                                                                                              MoveJ speed 60 deg/s, acceleration 80 deg/s^2 (useActiveTCP=true) feature=Base
                                                                                                Waypoint Waypoint_58: TCP in base x=365.318 y=-268.384 z=96.47 mm, rx=-1.8274 ry=-0.0328 rz=-0.0063 rad; joints [-29.465, -175.579, 2.323, 201.363, 146.436, -157.102] deg
                                                                                                URCap Gripper (Robotiq_Grippers, Robotiq Inc.) dataModel(position=0.0, force=0.0, speed=0.0, positionInDouble=0.0, forceInDouble=0.0, speedInDouble=0.0, slaveIds=[2], blocking=true)
                                                                                                MoveJ speed 60 deg/s, acceleration 80 deg/s^2 (useActiveTCP=true) feature=Base
                                                                                                  Waypoint Waypoint_2: motionParameters(jointSpeed=1.047198 jointAcceleration=1.396263 cartesianSpeed=0.25 cartesianAcceleration=1.2); TCP in base x=280.608 y=-116.08 z=398.046 mm, rx=-2.2371 ry=2.1464 rz=-0.0359 rad; joints [2.971, -88.172, -66.4, 247.256, 90.066, 0.681] deg
                                                                                                  MoveJ speed 60 deg/s, acceleration 80 deg/s^2 (useActiveTCP=true) feature=Base
                                                                                                    Waypoint Waypoint_56: TCP in base x=364.265 y=-116.054 z=192.334 mm, rx=-3.095 ry=0.0588 rz=0.0169 rad; joints [1.825, -110.55, -95.649, 295.749, 92.143, -86.362] deg
                                                                                                    URCap Gripper (Robotiq_Grippers, Robotiq Inc.) dataModel(position=100.0, force=0.0, speed=0.0, positionInDouble=100.0, forceInDouble=0.0, speedInDouble=0.0, slaveIds=[2], blocking=true)
                                                                                                    MoveJ speed 60 deg/s, acceleration 80 deg/s^2 (useActiveTCP=true) feature=Base
                                                                                                      Waypoint Waypoint_57: TCP in base x=364.254 y=-116.07 z=333.901 mm, rx=-3.0957 ry=-0.0405 rz=0.0191 rad; joints [1.801, -106.047, -62.68, 258.123, 92.053, -89.758] deg
                                                                                                      MoveJ speed 60 deg/s, acceleration 80 deg/s^2 (useActiveTCP=true) feature=Base
                                                                                                        Waypoint Waypoint_58: TCP in base x=365.318 y=-268.384 z=96.47 mm, rx=-1.8274 ry=-0.0328 rz=-0.0063 rad; joints [-29.465, -175.579, 2.323, 201.363, 146.436, -157.102] deg
                                                                                                        URCap Gripper (Robotiq_Grippers, Robotiq Inc.) dataModel(position=0.0, force=0.0, speed=0.0, positionInDouble=0.0, forceInDouble=0.0, speedInDouble=0.0, slaveIds=[2], blocking=true)
                                                                                                        MoveJ speed 60 deg/s, acceleration 80 deg/s^2 (useActiveTCP=true) feature=Base
                                                                                                          Waypoint Waypoint_2: motionParameters(jointSpeed=1.047198 jointAcceleration=1.396263 cartesianSpeed=0.25 cartesianAcceleration=1.2); TCP in base x=280.608 y=-116.08 z=398.046 mm, rx=-2.2371 ry=2.1464 rz=-0.0359 rad; joints [2.971, -88.172, -66.4, 247.256, 90.066, 0.681] deg
                                                                                                          Folder Mouvement D2
                                                                                                            MoveJ speed 60 deg/s, acceleration 80 deg/s^2 (useActiveTCP=true) feature=Base
                                                                                                              Waypoint Waypoint_2: motionParameters(jointSpeed=1.047198 jointAcceleration=1.396263 cartesianSpeed=0.25 cartesianAcceleration=1.2); TCP in base x=280.608 y=-116.08 z=398.046 mm, rx=-2.2371 ry=2.1464 rz=-0.0359 rad; joints [2.971, -88.172, -66.4, 247.256, 90.066, 0.681] deg
                                                                                                              MoveJ speed 60 deg/s, acceleration 80 deg/s^2 (useActiveTCP=true) feature=Base
                                                                                                                Waypoint Waypoint_56: TCP in base x=364.265 y=-116.054 z=192.334 mm, rx=-3.095 ry=0.0588 rz=0.0169 rad; joints [1.825, -110.55, -95.649, 295.749, 92.143, -86.362] deg
                                                                                                                URCap Gripper (Robotiq_Grippers, Robotiq Inc.) dataModel(position=100.0, force=0.0, speed=0.0, positionInDouble=100.0, forceInDouble=0.0, speedInDouble=0.0, slaveIds=[2], blocking=true)
                                                                                                                MoveJ speed 60 deg/s, acceleration 80 deg/s^2 (useActiveTCP=true) feature=Base
                                                                                                                  Waypoint Waypoint_57: TCP in base x=364.254 y=-116.07 z=333.901 mm, rx=-3.0957 ry=-0.0405 rz=0.0191 rad; joints [1.801, -106.047, -62.68, 258.123, 92.053, -89.758] deg
                                                                                                                  MoveJ speed 60 deg/s, acceleration 80 deg/s^2 (useActiveTCP=true) feature=Base
                                                                                                                    Waypoint Waypoint_58: TCP in base x=365.318 y=-268.384 z=96.47 mm, rx=-1.8274 ry=-0.0328 rz=-0.0063 rad; joints [-29.465, -175.579, 2.323, 201.363, 146.436, -157.102] deg
                                                                                                                    URCap Gripper (Robotiq_Grippers, Robotiq Inc.) dataModel(position=0.0, force=0.0, speed=0.0, positionInDouble=0.0, forceInDouble=0.0, speedInDouble=0.0, slaveIds=[2], blocking=true)
                                                                                                                    MoveJ speed 60 deg/s, acceleration 80 deg/s^2 (useActiveTCP=true) feature=Base
                                                                                                                      Waypoint Waypoint_2: motionParameters(jointSpeed=1.047198 jointAcceleration=1.396263 cartesianSpeed=0.25 cartesianAcceleration=1.2); TCP in base x=280.608 y=-116.08 z=398.046 mm, rx=-2.2371 ry=2.1464 rz=-0.0359 rad; joints [2.971, -88.172, -66.4, 247.256, 90.066, 0.681] deg
                                                                                                                      MoveJ speed 60 deg/s, acceleration 80 deg/s^2 (useActiveTCP=true) feature=Base
                                                                                                                        Waypoint Waypoint_56: TCP in base x=364.265 y=-116.054 z=192.334 mm, rx=-3.095 ry=0.0588 rz=0.0169 rad; joints [1.825, -110.55, -95.649, 295.749, 92.143, -86.362] deg
                                                                                                                        URCap Gripper (Robotiq_Grippers, Robotiq Inc.) dataModel(position=100.0, force=0.0, speed=0.0, positionInDouble=100.0, forceInDouble=0.0, speedInDouble=0.0, slaveIds=[2], blocking=true)
                                                                                                                        MoveJ speed 60 deg/s, acceleration 80 deg/s^2 (useActiveTCP=true) feature=Base
                                                                                                                          Waypoint Waypoint_57: TCP in base x=364.254 y=-116.07 z=333.901 mm, rx=-3.0957 ry=-0.0405 rz=0.0191 rad; joints [1.801, -106.047, -62.68, 258.123, 92.053, -89.758] deg
                                                                                                                          MoveJ speed 60 deg/s, acceleration 80 deg/s^2 (useActiveTCP=true) feature=Base
                                                                                                                            Waypoint Waypoint_58: TCP in base x=365.318 y=-268.384 z=96.47 mm, rx=-1.8274 ry=-0.0328 rz=-0.0063 rad; joints [-29.465, -175.579, 2.323, 201.363, 146.436, -157.102] deg
                                                                                                                            URCap Gripper (Robotiq_Grippers, Robotiq Inc.) dataModel(position=0.0, force=0.0, speed=0.0, positionInDouble=0.0, forceInDouble=0.0, speedInDouble=0.0, slaveIds=[2], blocking=true)
                                                                                                                            MoveJ speed 60 deg/s, acceleration 80 deg/s^2 (useActiveTCP=true) feature=Base
                                                                                                                              Waypoint Waypoint_2: motionParameters(jointSpeed=1.047198 jointAcceleration=1.396263 cartesianSpeed=0.25 cartesianAcceleration=1.2); TCP in base x=280.608 y=-116.08 z=398.046 mm, rx=-2.2371 ry=2.1464 rz=-0.0359 rad; joints [2.971, -88.172, -66.4, 247.256, 90.066, 0.681] deg
                                                                                                                              MoveJ speed 60 deg/s, acceleration 80 deg/s^2 (useActiveTCP=true) feature=Base
                                                                                                                                Waypoint Waypoint_59: TCP in base x=361.348 y=-116.091 z=193.172 mm, rx=-2.2553 ry=2.1644 rz=0.0052 rad; joints [2.324, -109.416, -97.451, 297.435, 90.248, -0.396] deg
                                                                                                                                URCap Gripper (Robotiq_Grippers, Robotiq Inc.) dataModel(position=100.0, force=0.0, speed=0.0, positionInDouble=100.0, forceInDouble=0.0, speedInDouble=0.0, slaveIds=[2], blocking=true)
                                                                                                                                MoveJ speed 60 deg/s, acceleration 80 deg/s^2 (useActiveTCP=true) feature=Base
                                                                                                                                  Waypoint Waypoint_63: TCP in base x=361.345 y=-116.096 z=193.168 mm, rx=2.0818 ry=2.2845 rz=0.0599 rad; joints [2.646, -108.789, -99.797, 302.251, 89.051, 176.908] deg
                                                                                                                                  URCap Gripper (Robotiq_Grippers, Robotiq Inc.) dataModel(position=0.0, force=0.0, speed=0.0, positionInDouble=0.0, forceInDouble=0.0, speedInDouble=0.0, slaveIds=[2], blocking=true)
                                                                                                                                  MoveJ speed 60 deg/s, acceleration 80 deg/s^2 (useActiveTCP=true) feature=Base
                                                                                                                                    Waypoint Waypoint_2: motionParameters(jointSpeed=1.047198 jointAcceleration=1.396263 cartesianSpeed=0.25 cartesianAcceleration=1.2); TCP in base x=280.608 y=-116.08 z=398.046 mm, rx=-2.2371 ry=2.1464 rz=-0.0359 rad; joints [2.971, -88.172, -66.4, 247.256, 90.066, 0.681] deg
                                                                                                                                    MoveJ speed 60 deg/s, acceleration 80 deg/s^2 (useActiveTCP=true) feature=Base
                                                                                                                                      Waypoint Waypoint_2: motionParameters(jointSpeed=1.047198 jointAcceleration=1.396263 cartesianSpeed=0.25 cartesianAcceleration=1.2); TCP in base x=280.608 y=-116.08 z=398.046 mm, rx=-2.2371 ry=2.1464 rz=-0.0359 rad; joints [2.971, -88.172, -66.4, 247.256, 90.066, 0.681] deg
                                                                                                                                      MoveJ speed 60 deg/s, acceleration 80 deg/s^2 (useActiveTCP=true) feature=Base
                                                                                                                                        Waypoint Waypoint_56: TCP in base x=364.265 y=-116.054 z=192.334 mm, rx=-3.095 ry=0.0588 rz=0.0169 rad; joints [1.825, -110.55, -95.649, 295.749, 92.143, -86.362] deg
                                                                                                                                        URCap Gripper (Robotiq_Grippers, Robotiq Inc.) dataModel(position=100.0, force=0.0, speed=0.0, positionInDouble=100.0, forceInDouble=0.0, speedInDouble=0.0, slaveIds=[2], blocking=true)
                                                                                                                                        MoveJ speed 60 deg/s, acceleration 80 deg/s^2 (useActiveTCP=true) feature=Base
                                                                                                                                          Waypoint Waypoint_57: TCP in base x=364.254 y=-116.07 z=333.901 mm, rx=-3.0957 ry=-0.0405 rz=0.0191 rad; joints [1.801, -106.047, -62.68, 258.123, 92.053, -89.758] deg
                                                                                                                                          MoveJ speed 60 deg/s, acceleration 80 deg/s^2 (useActiveTCP=true) feature=Base
                                                                                                                                            Waypoint Waypoint_58: TCP in base x=365.318 y=-268.384 z=96.47 mm, rx=-1.8274 ry=-0.0328 rz=-0.0063 rad; joints [-29.465, -175.579, 2.323, 201.363, 146.436, -157.102] deg
                                                                                                                                            URCap Gripper (Robotiq_Grippers, Robotiq Inc.) dataModel(position=0.0, force=0.0, speed=0.0, positionInDouble=0.0, forceInDouble=0.0, speedInDouble=0.0, slaveIds=[2], blocking=true)
                                                                                                                                            MoveJ speed 60 deg/s, acceleration 80 deg/s^2 (useActiveTCP=true) feature=Base
                                                                                                                                              Waypoint Waypoint_2: motionParameters(jointSpeed=1.047198 jointAcceleration=1.396263 cartesianSpeed=0.25 cartesianAcceleration=1.2); TCP in base x=280.608 y=-116.08 z=398.046 mm, rx=-2.2371 ry=2.1464 rz=-0.0359 rad; joints [2.971, -88.172, -66.4, 247.256, 90.066, 0.681] deg
                                                                                                                                              MoveJ speed 60 deg/s, acceleration 80 deg/s^2 (useActiveTCP=true) feature=Base
                                                                                                                                                Waypoint Waypoint_56: TCP in base x=364.265 y=-116.054 z=192.334 mm, rx=-3.095 ry=0.0588 rz=0.0169 rad; joints [1.825, -110.55, -95.649, 295.749, 92.143, -86.362] deg
                                                                                                                                                URCap Gripper (Robotiq_Grippers, Robotiq Inc.) dataModel(position=100.0, force=0.0, speed=0.0, positionInDouble=100.0, forceInDouble=0.0, speedInDouble=0.0, slaveIds=[2], blocking=true)
                                                                                                                                                MoveJ speed 60 deg/s, acceleration 80 deg/s^2 (useActiveTCP=true) feature=Base
                                                                                                                                                  Waypoint Waypoint_57: TCP in base x=364.254 y=-116.07 z=333.901 mm, rx=-3.0957 ry=-0.0405 rz=0.0191 rad; joints [1.801, -106.047, -62.68, 258.123, 92.053, -89.758] deg
                                                                                                                                                  MoveJ speed 60 deg/s, acceleration 80 deg/s^2 (useActiveTCP=true) feature=Base
                                                                                                                                                    Waypoint Waypoint_58: TCP in base x=365.318 y=-268.384 z=96.47 mm, rx=-1.8274 ry=-0.0328 rz=-0.0063 rad; joints [-29.465, -175.579, 2.323, 201.363, 146.436, -157.102] deg
                                                                                                                                                    URCap Gripper (Robotiq_Grippers, Robotiq Inc.) dataModel(position=0.0, force=0.0, speed=0.0, positionInDouble=0.0, forceInDouble=0.0, speedInDouble=0.0, slaveIds=[2], blocking=true)
                                                                                                                                                    MoveJ speed 60 deg/s, acceleration 80 deg/s^2 (useActiveTCP=true) feature=Base
                                                                                                                                                      Waypoint Waypoint_2: motionParameters(jointSpeed=1.047198 jointAcceleration=1.396263 cartesianSpeed=0.25 cartesianAcceleration=1.2); TCP in base x=280.608 y=-116.08 z=398.046 mm, rx=-2.2371 ry=2.1464 rz=-0.0359 rad; joints [2.971, -88.172, -66.4, 247.256, 90.066, 0.681] deg
